{attribute 'no_explicit_call' := 'Direct call is not allowed'} 
PROGRAM WideStringHelper
VAR_OUTPUT
	NewLine : WSTRING(1) := TO_WSTRING(Tc2_System.F_ToCHR(10)); 
END_VAR

METHOD AnyToString : WSTRING(255)
VAR_INPUT
	value : ANY;
END_VAR
AnyToString := InternalAnyToString(value);
END_METHOD

METHOD Append : BOOL
VAR_INPUT
	destinationString : ANY_STRING;
	sourceString : WSTRING(255);
END_VAR
VAR
	sources : ARRAY [1..1] OF POINTER TO WSTRING(255);
END_VAR
sources[1] := ADR(sourceString);

Append := InternalAppend(destinationString, sources);
END_METHOD

METHOD Append1 : BOOL
VAR_INPUT
	destinationString : ANY_STRING;
	sourceString1 : WSTRING(255);
END_VAR
VAR
	sources : ARRAY [1..1] OF POINTER TO WSTRING(255);
END_VAR
sources[1] := ADR(sourceString1);

Append1 := InternalAppend(destinationString, sources);
END_METHOD

METHOD Append10 : BOOL
VAR_INPUT
	destinationString : ANY_STRING;
	sourceString1 : WSTRING(255);
	sourceString2 : WSTRING(255);
	sourceString3 : WSTRING(255);
	sourceString4 : WSTRING(255);
	sourceString5 : WSTRING(255);
	sourceString6 : WSTRING(255);
	sourceString7 : WSTRING(255);
	sourceString8 : WSTRING(255);
	sourceString9 : WSTRING(255);
	sourceString10 : WSTRING(255);
END_VAR
VAR
	sources : ARRAY [1..10] OF POINTER TO WSTRING(255);
END_VAR
sources[1] := ADR(sourceString1);
sources[2] := ADR(sourceString2);
sources[3] := ADR(sourceString3);
sources[4] := ADR(sourceString4);
sources[5] := ADR(sourceString5);
sources[6] := ADR(sourceString6);
sources[7] := ADR(sourceString7);
sources[8] := ADR(sourceString8);
sources[9] := ADR(sourceString9);
sources[10] := ADR(sourceString10);

Append10 := InternalAppend(destinationString, sources);
END_METHOD

METHOD Append11 : BOOL
VAR_INPUT
	destinationString : ANY_STRING;
	sourceString1 : WSTRING(255);
	sourceString2 : WSTRING(255);
	sourceString3 : WSTRING(255);
	sourceString4 : WSTRING(255);
	sourceString5 : WSTRING(255);
	sourceString6 : WSTRING(255);
	sourceString7 : WSTRING(255);
	sourceString8 : WSTRING(255);
	sourceString9 : WSTRING(255);
	sourceString10 : WSTRING(255);
	sourceString11 : WSTRING(255);
END_VAR
VAR
	sources : ARRAY [1..11] OF POINTER TO WSTRING(255);
END_VAR
sources[1] := ADR(sourceString1);
sources[2] := ADR(sourceString2);
sources[3] := ADR(sourceString3);
sources[4] := ADR(sourceString4);
sources[5] := ADR(sourceString5);
sources[6] := ADR(sourceString6);
sources[7] := ADR(sourceString7);
sources[8] := ADR(sourceString8);
sources[9] := ADR(sourceString9);
sources[10] := ADR(sourceString10);
sources[11] := ADR(sourceString11);

Append11 := InternalAppend(destinationString, sources);
END_METHOD

METHOD Append12 : BOOL
VAR_INPUT
	destinationString : ANY_STRING;
	sourceString1 : WSTRING(255);
	sourceString2 : WSTRING(255);
	sourceString3 : WSTRING(255);
	sourceString4 : WSTRING(255);
	sourceString5 : WSTRING(255);
	sourceString6 : WSTRING(255);
	sourceString7 : WSTRING(255);
	sourceString8 : WSTRING(255);
	sourceString9 : WSTRING(255);
	sourceString10 : WSTRING(255);
	sourceString11 : WSTRING(255);
	sourceString12 : WSTRING(255);
END_VAR
VAR
	sources : ARRAY [1..12] OF POINTER TO WSTRING(255);
END_VAR
sources[1] := ADR(sourceString1);
sources[2] := ADR(sourceString2);
sources[3] := ADR(sourceString3);
sources[4] := ADR(sourceString4);
sources[5] := ADR(sourceString5);
sources[6] := ADR(sourceString6);
sources[7] := ADR(sourceString7);
sources[8] := ADR(sourceString8);
sources[9] := ADR(sourceString9);
sources[10] := ADR(sourceString10);
sources[11] := ADR(sourceString11);
sources[12] := ADR(sourceString12);

Append12 := InternalAppend(destinationString, sources);
END_METHOD

METHOD Append13 : BOOL
VAR_INPUT
	destinationString : ANY_STRING;
	sourceString1 : WSTRING(255);
	sourceString2 : WSTRING(255);
	sourceString3 : WSTRING(255);
	sourceString4 : WSTRING(255);
	sourceString5 : WSTRING(255);
	sourceString6 : WSTRING(255);
	sourceString7 : WSTRING(255);
	sourceString8 : WSTRING(255);
	sourceString9 : WSTRING(255);
	sourceString10 : WSTRING(255);
	sourceString11 : WSTRING(255);
	sourceString12 : WSTRING(255);
	sourceString13 : WSTRING(255);
END_VAR
VAR
	sources : ARRAY [1..13] OF POINTER TO WSTRING(255);
END_VAR
sources[1] := ADR(sourceString1);
sources[2] := ADR(sourceString2);
sources[3] := ADR(sourceString3);
sources[4] := ADR(sourceString4);
sources[5] := ADR(sourceString5);
sources[6] := ADR(sourceString6);
sources[7] := ADR(sourceString7);
sources[8] := ADR(sourceString8);
sources[9] := ADR(sourceString9);
sources[10] := ADR(sourceString10);
sources[11] := ADR(sourceString11);
sources[12] := ADR(sourceString12);
sources[13] := ADR(sourceString13);

Append13 := InternalAppend(destinationString, sources);
END_METHOD

METHOD Append14 : BOOL
VAR_INPUT
	destinationString : ANY_STRING;
	sourceString1 : WSTRING(255);
	sourceString2 : WSTRING(255);
	sourceString3 : WSTRING(255);
	sourceString4 : WSTRING(255);
	sourceString5 : WSTRING(255);
	sourceString6 : WSTRING(255);
	sourceString7 : WSTRING(255);
	sourceString8 : WSTRING(255);
	sourceString9 : WSTRING(255);
	sourceString10 : WSTRING(255);
	sourceString11 : WSTRING(255);
	sourceString12 : WSTRING(255);
	sourceString13 : WSTRING(255);
	sourceString14 : WSTRING(255);
END_VAR
VAR
	sources : ARRAY [1..14] OF POINTER TO WSTRING(255);
END_VAR
sources[1] := ADR(sourceString1);
sources[2] := ADR(sourceString2);
sources[3] := ADR(sourceString3);
sources[4] := ADR(sourceString4);
sources[5] := ADR(sourceString5);
sources[6] := ADR(sourceString6);
sources[7] := ADR(sourceString7);
sources[8] := ADR(sourceString8);
sources[9] := ADR(sourceString9);
sources[10] := ADR(sourceString10);
sources[11] := ADR(sourceString11);
sources[12] := ADR(sourceString12);
sources[13] := ADR(sourceString13);
sources[14] := ADR(sourceString14);

Append14 := InternalAppend(destinationString, sources);
END_METHOD

METHOD Append2 : BOOL
VAR_INPUT
	destinationString : ANY_STRING;
	sourceString1 : WSTRING(255);
	sourceString2 : WSTRING(255);
END_VAR
VAR
	sources : ARRAY [1..2] OF POINTER TO WSTRING(255);
END_VAR
sources[1] := ADR(sourceString1);
sources[2] := ADR(sourceString2);

Append2 := InternalAppend(destinationString, sources);
END_METHOD

METHOD Append3 : BOOL
VAR_INPUT
	destinationString : ANY_STRING;
	sourceString1 : WSTRING(255);
	sourceString2 : WSTRING(255);
	sourceString3 : WSTRING(255);
END_VAR
VAR
	sources : ARRAY [1..3] OF POINTER TO WSTRING(255);
END_VAR
sources[1] := ADR(sourceString1);
sources[2] := ADR(sourceString2);
sources[3] := ADR(sourceString3);

Append3 := InternalAppend(destinationString, sources);
END_METHOD

METHOD Append4 : BOOL
VAR_INPUT
	destinationString : ANY_STRING;
	sourceString1 : WSTRING(255);
	sourceString2 : WSTRING(255);
	sourceString3 : WSTRING(255);
	sourceString4 : WSTRING(255);
END_VAR
VAR
	sources : ARRAY [1..4] OF POINTER TO WSTRING(255);
END_VAR
sources[1] := ADR(sourceString1);
sources[2] := ADR(sourceString2);
sources[3] := ADR(sourceString3);
sources[4] := ADR(sourceString4);

Append4 := InternalAppend(destinationString, sources);
END_METHOD

METHOD Append5 : BOOL
VAR_INPUT
	destinationString : ANY_STRING;
	sourceString1 : WSTRING(255);
	sourceString2 : WSTRING(255);
	sourceString3 : WSTRING(255);
	sourceString4 : WSTRING(255);
	sourceString5 : WSTRING(255);
END_VAR
VAR
	sources : ARRAY [1..5] OF POINTER TO WSTRING(255);
END_VAR
sources[1] := ADR(sourceString1);
sources[2] := ADR(sourceString2);
sources[3] := ADR(sourceString3);
sources[4] := ADR(sourceString4);
sources[5] := ADR(sourceString5);

Append5 := InternalAppend(destinationString, sources);
END_METHOD

METHOD Append6 : BOOL
VAR_INPUT
	destinationString : ANY_STRING;
	sourceString1 : WSTRING(255);
	sourceString2 : WSTRING(255);
	sourceString3 : WSTRING(255);
	sourceString4 : WSTRING(255);
	sourceString5 : WSTRING(255);
	sourceString6 : WSTRING(255);
END_VAR
VAR
	sources : ARRAY [1..6] OF POINTER TO WSTRING(255);
END_VAR
sources[1] := ADR(sourceString1);
sources[2] := ADR(sourceString2);
sources[3] := ADR(sourceString3);
sources[4] := ADR(sourceString4);
sources[5] := ADR(sourceString5);
sources[6] := ADR(sourceString6);

Append6 := InternalAppend(destinationString, sources);
END_METHOD

METHOD Append7 : BOOL
VAR_INPUT
	destinationString : ANY_STRING;
	sourceString1 : WSTRING(255);
	sourceString2 : WSTRING(255);
	sourceString3 : WSTRING(255);
	sourceString4 : WSTRING(255);
	sourceString5 : WSTRING(255);
	sourceString6 : WSTRING(255);
	sourceString7 : WSTRING(255);
END_VAR
VAR
	sources : ARRAY [1..7] OF POINTER TO WSTRING(255);
END_VAR
sources[1] := ADR(sourceString1);
sources[2] := ADR(sourceString2);
sources[3] := ADR(sourceString3);
sources[4] := ADR(sourceString4);
sources[5] := ADR(sourceString5);
sources[6] := ADR(sourceString6);
sources[7] := ADR(sourceString7);

Append7 := InternalAppend(destinationString, sources);
END_METHOD

METHOD Append8 : BOOL
VAR_INPUT
	destinationString : ANY_STRING;
	sourceString1 : WSTRING(255);
	sourceString2 : WSTRING(255);
	sourceString3 : WSTRING(255);
	sourceString4 : WSTRING(255);
	sourceString5 : WSTRING(255);
	sourceString6 : WSTRING(255);
	sourceString7 : WSTRING(255);
	sourceString8 : WSTRING(255);
END_VAR
VAR
	sources : ARRAY [1..8] OF POINTER TO WSTRING(255);
END_VAR
sources[1] := ADR(sourceString1);
sources[2] := ADR(sourceString2);
sources[3] := ADR(sourceString3);
sources[4] := ADR(sourceString4);
sources[5] := ADR(sourceString5);
sources[6] := ADR(sourceString6);
sources[7] := ADR(sourceString7);
sources[8] := ADR(sourceString8);

Append8 := InternalAppend(destinationString, sources);
END_METHOD

METHOD Append9 : BOOL
VAR_INPUT
	destinationString : ANY_STRING;
	sourceString1 : WSTRING(255);
	sourceString2 : WSTRING(255);
	sourceString3 : WSTRING(255);
	sourceString4 : WSTRING(255);
	sourceString5 : WSTRING(255);
	sourceString6 : WSTRING(255);
	sourceString7 : WSTRING(255);
	sourceString8 : WSTRING(255);
	sourceString9 : WSTRING(255);
END_VAR
VAR
	sources : ARRAY [1..9] OF POINTER TO WSTRING(255);
END_VAR
sources[1] := ADR(sourceString1);
sources[2] := ADR(sourceString2);
sources[3] := ADR(sourceString3);
sources[4] := ADR(sourceString4);
sources[5] := ADR(sourceString5);
sources[6] := ADR(sourceString6);
sources[7] := ADR(sourceString7);
sources[8] := ADR(sourceString8);
sources[9] := ADR(sourceString9);

Append9 := InternalAppend(destinationString, sources);
END_METHOD

METHOD Concat10 : WSTRING(255)
VAR_INPUT
	string1 : WSTRING(255);
	string2 : WSTRING(255);
	string3 : WSTRING(255);
	string4 : WSTRING(255);
	string5 : WSTRING(255);
	string6 : WSTRING(255);
	string7 : WSTRING(255);
	string8 : WSTRING(255);
	string9 : WSTRING(255);
	string10 : WSTRING(255);
END_VAR
Concat10 := Tc2_Standard.WCONCAT(
	Tc2_Standard.WCONCAT(
		Tc2_Standard.WCONCAT(Tc2_Standard.WCONCAT(string1, string2), Tc2_Standard.WCONCAT(string3, string4)), 
		Tc2_Standard.WCONCAT(Tc2_Standard.WCONCAT(string5, string6), Tc2_Standard.WCONCAT(string7, string8)) 
	),
	Tc2_Standard.WCONCAT(string9, string10));
END_METHOD

METHOD Concat11 : WSTRING(255)
VAR_INPUT
	string1 : WSTRING(255);
	string2 : WSTRING(255);
	string3 : WSTRING(255);
	string4 : WSTRING(255);
	string5 : WSTRING(255);
	string6 : WSTRING(255);
	string7 : WSTRING(255);
	string8 : WSTRING(255);
	string9 : WSTRING(255);
	string10 : WSTRING(255);
	string11 : WSTRING(255);
END_VAR
Concat11 := Tc2_Standard.WCONCAT(
	Tc2_Standard.WCONCAT(
		Tc2_Standard.WCONCAT(Tc2_Standard.WCONCAT(string1, string2), Tc2_Standard.WCONCAT(string3, string4)), 
		Tc2_Standard.WCONCAT(Tc2_Standard.WCONCAT(string5, string6), Tc2_Standard.WCONCAT(string7, string8)) 
	),
	Tc2_Standard.WCONCAT(
		Tc2_Standard.WCONCAT(string9, string10),
		string11
	)
);
END_METHOD

METHOD Concat12 : WSTRING(255)
VAR_INPUT
	string1 : WSTRING(255);
	string2 : WSTRING(255);
	string3 : WSTRING(255);
	string4 : WSTRING(255);
	string5 : WSTRING(255);
	string6 : WSTRING(255);
	string7 : WSTRING(255);
	string8 : WSTRING(255);
	string9 : WSTRING(255);
	string10 : WSTRING(255);
	string11 : WSTRING(255);
	string12 : WSTRING(255);
END_VAR
Concat12 := Tc2_Standard.WCONCAT(
	Tc2_Standard.WCONCAT(
		Tc2_Standard.WCONCAT(Tc2_Standard.WCONCAT(string1, string2), Tc2_Standard.WCONCAT(string3, string4)), 
		Tc2_Standard.WCONCAT(Tc2_Standard.WCONCAT(string5, string6), Tc2_Standard.WCONCAT(string7, string8)) 
	),
	Tc2_Standard.WCONCAT(
		Tc2_Standard.WCONCAT(string9, string10),
		Tc2_Standard.WCONCAT(string11, string12)
	)
);
END_METHOD

METHOD Concat13 : WSTRING(255)
VAR_INPUT
	string1 : WSTRING(255);
	string2 : WSTRING(255);
	string3 : WSTRING(255);
	string4 : WSTRING(255);
	string5 : WSTRING(255);
	string6 : WSTRING(255);
	string7 : WSTRING(255);
	string8 : WSTRING(255);
	string9 : WSTRING(255);
	string10 : WSTRING(255);
	string11 : WSTRING(255);
	string12 : WSTRING(255);
	string13 : WSTRING(255);
END_VAR
Concat13 := Tc2_Standard.WCONCAT(
	Tc2_Standard.WCONCAT(
		Tc2_Standard.WCONCAT(Tc2_Standard.WCONCAT(string1, string2), Tc2_Standard.WCONCAT(string3, string4)), 
		Tc2_Standard.WCONCAT(Tc2_Standard.WCONCAT(string5, string6), Tc2_Standard.WCONCAT(string7, string8)) 
	),
	Tc2_Standard.WCONCAT(
		Tc2_Standard.WCONCAT(Tc2_Standard.WCONCAT(string9, string10), Tc2_Standard.WCONCAT(string11, string12)),
		string13
	)
);
END_METHOD

METHOD Concat14 : WSTRING(255)
VAR_INPUT
	string1 : WSTRING(255);
	string2 : WSTRING(255);
	string3 : WSTRING(255);
	string4 : WSTRING(255);
	string5 : WSTRING(255);
	string6 : WSTRING(255);
	string7 : WSTRING(255);
	string8 : WSTRING(255);
	string9 : WSTRING(255);
	string10 : WSTRING(255);
	string11 : WSTRING(255);
	string12 : WSTRING(255);
	string13 : WSTRING(255);
	string14 : WSTRING(255);
END_VAR
Concat14 := Tc2_Standard.WCONCAT(
	Tc2_Standard.WCONCAT(
		Tc2_Standard.WCONCAT(Tc2_Standard.WCONCAT(string1, string2), Tc2_Standard.WCONCAT(string3, string4)), 
		Tc2_Standard.WCONCAT(Tc2_Standard.WCONCAT(string5, string6), Tc2_Standard.WCONCAT(string7, string8)) 
	),
	Tc2_Standard.WCONCAT(
		Tc2_Standard.WCONCAT(Tc2_Standard.WCONCAT(string9, string10), Tc2_Standard.WCONCAT(string11, string12)),
		Tc2_Standard.WCONCAT(string13, string14)
	)
);
END_METHOD

METHOD Concat2 : WSTRING(255)
VAR_INPUT
	string1 : WSTRING(255);
	string2 : WSTRING(255);
END_VAR
Concat2 := Tc2_Standard.WCONCAT(string1, string2);
END_METHOD

METHOD Concat3 : WSTRING(255)
VAR_INPUT
	string1 : WSTRING(255);
	string2 : WSTRING(255);
	string3 : WSTRING(255);
END_VAR
Concat3 := Tc2_Standard.WCONCAT(Tc2_Standard.WCONCAT(string1, string2), string3);
END_METHOD

METHOD Concat4 : WSTRING(255)
VAR_INPUT
	string1 : WSTRING(255);
	string2 : WSTRING(255);
	string3 : WSTRING(255);
	string4 : WSTRING(255);
END_VAR
Concat4 := Tc2_Standard.WCONCAT(Tc2_Standard.WCONCAT(string1, string2), Tc2_Standard.WCONCAT(string3, string4));
END_METHOD

METHOD Concat5 : WSTRING(255)
VAR_INPUT
	string1 : WSTRING(255);
	string2 : WSTRING(255);
	string3 : WSTRING(255);
	string4 : WSTRING(255);
	string5 : WSTRING(255);
END_VAR
Concat5 := Tc2_Standard.WCONCAT(Tc2_Standard.WCONCAT(Tc2_Standard.WCONCAT(string1, string2), Tc2_Standard.WCONCAT(string3, string4)), string5);
END_METHOD

METHOD Concat6 : WSTRING(255)
VAR_INPUT
	string1 : WSTRING(255);
	string2 : WSTRING(255);
	string3 : WSTRING(255);
	string4 : WSTRING(255);
	string5 : WSTRING(255);
	string6 : WSTRING(255);
END_VAR
Concat6 := Tc2_Standard.WCONCAT(
	Tc2_Standard.WCONCAT(Tc2_Standard.WCONCAT(string1, string2), Tc2_Standard.WCONCAT(string3, string4)), 
	Tc2_Standard.WCONCAT(string5, string6)
);
END_METHOD

METHOD Concat7 : WSTRING(255)
VAR_INPUT
	string1 : WSTRING(255);
	string2 : WSTRING(255);
	string3 : WSTRING(255);
	string4 : WSTRING(255);
	string5 : WSTRING(255);
	string6 : WSTRING(255);
	string7 : WSTRING(255);
END_VAR
Concat7 := Tc2_Standard.WCONCAT(
	Tc2_Standard.WCONCAT(Tc2_Standard.WCONCAT(string1, string2), Tc2_Standard.WCONCAT(string3, string4)), 
	Tc2_Standard.WCONCAT(Tc2_Standard.WCONCAT(string5, string6), string7)
);
END_METHOD

METHOD Concat8 : WSTRING(255)
VAR_INPUT
	string1 : WSTRING(255);
	string2 : WSTRING(255);
	string3 : WSTRING(255);
	string4 : WSTRING(255);
	string5 : WSTRING(255);
	string6 : WSTRING(255);
	string7 : WSTRING(255);
	string8 : WSTRING(255);
END_VAR
Concat8 := Tc2_Standard.WCONCAT(
	Tc2_Standard.WCONCAT(Tc2_Standard.WCONCAT(string1, string2), Tc2_Standard.WCONCAT(string3, string4)), 
	Tc2_Standard.WCONCAT(Tc2_Standard.WCONCAT(string5, string6), Tc2_Standard.WCONCAT(string7, string8)) 
);
END_METHOD

METHOD Concat9 : WSTRING(255)
VAR_INPUT
	string1 : WSTRING(255);
	string2 : WSTRING(255);
	string3 : WSTRING(255);
	string4 : WSTRING(255);
	string5 : WSTRING(255);
	string6 : WSTRING(255);
	string7 : WSTRING(255);
	string8 : WSTRING(255);
	string9 : WSTRING(255);
END_VAR
Concat9 := Tc2_Standard.WCONCAT(
	Tc2_Standard.WCONCAT(
		Tc2_Standard.WCONCAT(Tc2_Standard.WCONCAT(string1, string2), Tc2_Standard.WCONCAT(string3, string4)), 
		Tc2_Standard.WCONCAT(Tc2_Standard.WCONCAT(string5, string6), Tc2_Standard.WCONCAT(string7, string8)) 
	),
	string9);
END_METHOD

METHOD DateAndTimeToString : WSTRING
VAR_INPUT
	value : DATE_AND_TIME;
	dateValuesSeparator : STRING(1) := '_';
	dateAndTimeSeparator : STRING(1) := '-';
	timeValuesSeparator : STRING(1) := '_';
END_VAR
VAR
	result : STRING;
END_VAR
result := TO_STRING(value);

result := Tc2_Standard.DELETE(result, 3, 1);

result := Tc2_Standard.REPLACE(result, dateValuesSeparator, 1, 5);
result := Tc2_Standard.REPLACE(result, dateValuesSeparator, 1, 8);
result := Tc2_Standard.REPLACE(result, dateAndTimeSeparator, 1, 11);
result := Tc2_Standard.REPLACE(result, timeValuesSeparator, 1, 14);
result := Tc2_Standard.REPLACE(result, timeValuesSeparator, 1, 17);

DateAndTimeToString := TO_WSTRING(result);
END_METHOD

METHOD INTERNAL InternalAnyToString : WSTRING(255)
VAR_INPUT
	value : __System.AnyType;
END_VAR
VAR
	anyBool : POINTER TO BOOL;

	anyByte : POINTER TO BYTE;
	anyWord : POINTER TO WORD;
	anyDWord : POINTER TO LWORD;
	anyLWord : POINTER TO LWORD;
	
	anySInt : POINTER TO SINT;
	anyInt : POINTER TO INT;
	anyDInt : POINTER TO DINT;
	anyLInt : POINTER TO LINT;
	
	anyUSInt : POINTER TO USINT;
	anyUInt : POINTER TO UINT;
	anyUDInt : POINTER TO UDINT;
	anyULInt : POINTER TO ULINT;
	
	anyReal : POINTER TO REAL;
	anyLReal : POINTER TO LREAL;

	anyString : POINTER TO STRING(255);
	anyWString : POINTER TO WSTRING(255);
	
	anyTime : POINTER TO TIME;
	anyLTime : POINTER TO LTIME;
	anyDate : POINTER TO DATE;
	anyDateAndTime : POINTER TO DATE_AND_TIME;
	anyTimeOfDay : POINTER TO TOD;
END_VAR
CASE value.TypeClass OF
	__SYSTEM.TYPE_CLASS.TYPE_BOOL:
		anyBool := value.pValue;
		InternalAnyToString := TO_WSTRING(anyBool^);		
	
	__SYSTEM.TYPE_CLASS.TYPE_BIT:
		anyByte := value.pValue;
		IF anyByte^ > 0 THEN
			InternalAnyToString := "1";		
		ELSE
			InternalAnyToString := "0";		
		END_IF
	
	__SYSTEM.TYPE_CLASS.TYPE_BYTE:
		anyByte := value.pValue;
		InternalAnyToString := TO_WSTRING(anyByte^);		
	__SYSTEM.TYPE_CLASS.TYPE_WORD:
		anyWord := value.pValue;
		InternalAnyToString := TO_WSTRING(anyWord^);
	__SYSTEM.TYPE_CLASS.TYPE_DWORD:
		anyDWord := value.pValue;
		InternalAnyToString := TO_WSTRING(anyDWord^);
	__SYSTEM.TYPE_CLASS.TYPE_LWORD:
		anyLWord := value.pValue;
		InternalAnyToString := TO_WSTRING(anyLWord^);
		
	__SYSTEM.TYPE_CLASS.TYPE_SINT:
		anySInt := value.pValue;
		InternalAnyToString := TO_WSTRING(anySInt^);
	__SYSTEM.TYPE_CLASS.TYPE_INT:
		anyInt := value.pValue;
		InternalAnyToString := TO_WSTRING(anyInt^);		
	__SYSTEM.TYPE_CLASS.TYPE_DINT:
		anyDInt := value.pValue;
		InternalAnyToString := TO_WSTRING(anyDInt^);
	__SYSTEM.TYPE_CLASS.TYPE_LINT:
		anyLInt := value.pValue;
		InternalAnyToString := TO_WSTRING(anyLInt^);
		
	__SYSTEM.TYPE_CLASS.TYPE_USINT:
		anyUSInt := value.pValue;
		InternalAnyToString := TO_WSTRING(anyUSInt^);
	__SYSTEM.TYPE_CLASS.TYPE_UINT:
		anyUInt := value.pValue;
		InternalAnyToString := TO_WSTRING(anyUInt^);		
	__SYSTEM.TYPE_CLASS.TYPE_UDINT:
		anyUDInt := value.pValue;
		InternalAnyToString := TO_WSTRING(anyUDInt^);
	__SYSTEM.TYPE_CLASS.TYPE_ULINT:
		anyULInt := value.pValue;
		InternalAnyToString := TO_WSTRING(anyULInt^);

	__SYSTEM.TYPE_CLASS.TYPE_REAL:
		anyReal := value.pValue;
		InternalAnyToString := TO_WSTRING(anyReal^);
	__SYSTEM.TYPE_CLASS.TYPE_LREAL:
		anyLReal := value.pValue;
		InternalAnyToString := TO_WSTRING(anyLReal^);
	
	__SYSTEM.TYPE_CLASS.TYPE_STRING:
		anyString := value.pValue;
		InternalAnyToString := TO_WSTRING(anyString^);
	__SYSTEM.TYPE_CLASS.TYPE_WSTRING:
		anyWString := value.pValue;
		InternalAnyToString := anyWString^;
	
	__SYSTEM.TYPE_CLASS.TYPE_TIME:
		anyTime := value.pValue;
		InternalAnyToString := TO_WSTRING(anyTime^);
	__SYSTEM.TYPE_CLASS.TYPE_LTIME:
		anyLTime := value.pValue;
		InternalAnyToString := TO_WSTRING(anyLTime^);
	__SYSTEM.TYPE_CLASS.TYPE_DATE:
		anyDate := value.pValue;
		InternalAnyToString := TO_WSTRING(anyDate^);
	__SYSTEM.TYPE_CLASS.TYPE_DATEANDTIME:
		anyDateAndTime := value.pValue;
		InternalAnyToString := TO_WSTRING(anyDateAndTime^);  
	__SYSTEM.TYPE_CLASS.TYPE_TIMEOFDAY:
		anyTimeOfDay := value.pValue;
		InternalAnyToString := TO_WSTRING(anyTimeOfDay^);
	
	__SYSTEM.TYPE_CLASS.TYPE_POINTER, __SYSTEM.TYPE_CLASS.TYPE_REFERENCE:
		InternalAnyToString := TO_WSTRING(Tc2_Utilities.PVOID_TO_HEXSTR(anyDate, 8, FALSE));		
	
	(*__SYSTEM.TYPE_CLASS.TYPE_SUBRANGE:
	__SYSTEM.TYPE_CLASS.TYPE_ENUM:
	__SYSTEM.TYPE_CLASS.TYPE_ARRAY:
	__SYSTEM.TYPE_CLASS.TYPE_PARAMS:
	__SYSTEM.TYPE_CLASS.TYPE_USERDEF:
	__SYSTEM.TYPE_CLASS.TYPE_NONE:
	__SYSTEM.TYPE_CLASS.TYPE_ANY:
	__SYSTEM.TYPE_CLASS.TYPE_ANYBIT:
	__SYSTEM.TYPE_CLASS.TYPE_ANYDATE:
	__SYSTEM.TYPE_CLASS.TYPE_ANYINT:
	__SYSTEM.TYPE_CLASS.TYPE_ANYNUM:
	__SYSTEM.TYPE_CLASS.TYPE_ANYREAL:
	__SYSTEM.TYPE_CLASS.TYPE_LAZY:
	__SYSTEM.TYPE_CLASS.TYPE_BITCONST:*)
	ELSE
		IF value.pValue <> 0 THEN
			InternalAnyToString := TO_WSTRING(value.pValue^); 
		ELSE
			InternalAnyToString := "NULL";
		END_IF
END_CASE
END_METHOD

METHOD INTERNAL InternalAppend : BOOL
VAR_INPUT
	destinationString : __SYSTEM.AnyType;
END_VAR
VAR_IN_OUT
	sourceStrings : ARRAY [*] OF POINTER TO WSTRING(255);
END_VAR
VAR
	i : DINT;
END_VAR
IF destinationString.TypeClass <> __SYSTEM.TYPE_CLASS.TYPE_WSTRING THEN
	RETURN;
END_IF	

FOR i := LOWER_BOUND(sourceStrings, 1) TO UPPER_BOUND(sourceStrings, 1) DO
	InternalAppend := Tc2_Utilities.WCONCAT2(destinationString.pValue, sourceStrings[i], destinationString.pValue, TO_UDINT(destinationString.diSize));	
END_FOR
END_METHOD

END_PROGRAM

(* stored: Version 1.1.0.1
   POU WideStringHelper: Id {f2b62380-bf78-436f-91e7-3a8440654572}, SpecialFunc None
   Folder Service members: Id {1ecfbf1d-7d0e-4566-abbe-72e054ea0151}
   Method AnyToString: Id {17d38b2c-68d3-4c9b-bfdc-5b5dcbc0e3da}
   Method Append: Id {0abbeab1-87d6-445a-be7e-01028a2ee5d0}
   Method Append1: Id {8ae54d0a-d199-4ca5-bf1a-a8dc731fbbed}
   Method Append10: Id {106fd8f3-40e3-49ce-be34-e9479f5ee394}
   Method Append11: Id {644a0f0e-2a23-4b37-9fd4-a5d2202bd213}
   Method Append12: Id {b9cb490d-cc36-4845-abc9-daa49db194d5}
   Method Append13: Id {e23ffdb6-afbd-44c5-ac8c-bd29f56db185}
   Method Append14: Id {05124919-d825-4d99-b37e-7b43602ef124}
   Method Append2: Id {f2762a28-ba20-4da3-bca6-4d7342e6ccc1}
   Method Append3: Id {a901e39c-74fb-456f-83c3-b55c09434265}
   Method Append4: Id {f16e517b-f218-46a2-baa0-b252e491b074}
   Method Append5: Id {651a3a52-6221-4a6d-9676-2c7128c556a2}
   Method Append6: Id {074d6c00-dbe9-4615-9fd1-f2449fdc2a24}
   Method Append7: Id {04973c34-3a08-42d5-b49e-39954c059a1b}
   Method Append8: Id {d3392a59-5d67-447b-87b7-7441a30a6c20}
   Method Append9: Id {69e07324-e292-4e35-b75f-e817eae7fe3d}
   Method Concat10: Id {89b82cd9-1fd4-40f4-a7bf-209c61b7f6cb}
   Method Concat11: Id {a768c2fd-1017-4225-89f8-dbb808006f68}
   Method Concat12: Id {356972f6-e7e0-4152-9e97-4a2502151e80}
   Method Concat13: Id {7fd72f1a-0293-4f99-9eb9-70aa83b15ff3}
   Method Concat14: Id {bb16bd0b-9d43-437e-84b2-c2ebcebe1eb9}
   Method Concat2: Id {b8d3f2d7-a38f-491f-9402-790706d9ac79}
   Method Concat3: Id {6cc4b694-bfce-4edf-a6b8-2346ef5e80aa}
   Method Concat4: Id {23030920-973f-4f7d-80e9-16dfaa2e863f}
   Method Concat5: Id {9e627e26-0dc8-48d9-b4cc-613b78b1dafc}
   Method Concat6: Id {989ef56c-493e-4d5b-beff-878d0e2b2e80}
   Method Concat7: Id {ffebfbe9-4a52-41a4-b954-94152957962e}
   Method Concat8: Id {489abba0-c5f9-46ee-82fb-dd6d8898d149}
   Method Concat9: Id {2215b580-dda9-47e9-b0b2-3e2a16a4eaa2}
   Method DateAndTimeToString: Id {2dbf6889-ac63-40bb-b159-7f5bcda0d03e}
   Method InternalAnyToString: Id {6abee510-4ede-4ea2-b6f7-c6402af23390}
   Method InternalAppend: Id {993a8ebe-26f7-4860-9a90-ac8cc45da36c} *)
